SUBAPPLICATION SubApp_PC_A (* Geraet A (Station 11, 192.168.1.11): 2 SoftKeys (Set/Reset) und GreenWhiteBackground am Set-SoftKey - 'SUB style', das Protokoll steckt im MyLib::sys-Composite (SoftKeySR_PC_A_OPC_Adapter), nicht in der Resource des Geraets - Adapter-Variante von Training_05, gleiche OPC-UA-Adressen *)
  (* Standard: 61499-2; Description: Copyright (c) 2026 Meisterschulen am Ostbahnhof This program and the accompanying materials are made available under the terms of the Eclipse Public License 2.0 which is available at https://www.eclipse.org/legal/epl-2.0/ SPDX-License-Identifier: EPL-2.0 *)
  (* Version 1.0, 2026-09-04, Franz Höpfinger, Meisterschulen am Ostbahnhof, initial API and implementation and/or initial documentation *)
  PACKAGE subapp::Training_07_OPC_UA_RES;
  IMPORT Uebungen::const::UT::DefaultPool::SoftKey_F1;
  IMPORT Uebungen::const::UT::DefaultPool::SoftKey_F2;
  IMPORT VV::const::OPC_UA::myOpcUaAddresses::SR2_SET_REMOTE_CALL;
  IMPORT VV::const::OPC_UA::myOpcUaAddresses::SR2_RESET_REMOTE_CALL;
  IMPORT VV::const::OPC_UA::myOpcUaAddresses::SR2_STATE_LOCAL_READ;
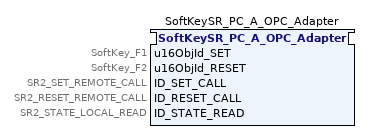
  SUBAPPS
    SoftKeySR_PC_A_OPC_Adapter : MyLib::sys::SoftKeySR_PC_A_OPC_Adapter(u16ObjId_SET := SoftKey_F1, u16ObjId_RESET := SoftKey_F2, ID_SET_CALL := SR2_SET_REMOTE_CALL, ID_RESET_CALL := SR2_RESET_REMOTE_CALL, ID_STATE_READ := SR2_STATE_LOCAL_READ);
  END_SUBAPPS
END_SUBAPPLICATION
